ABB RobotStudio station: Final_BT19MEC092_20211026-093550.rsstn

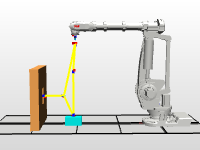
Station Solution1 (saved by RobotStudio 6.8.8307.1040)
Controller System1
  mechanical unit ROB_1: IRB6660_100_335__01, 6 joints, base frame (0, 0, 0) mm
Layout (positions relative to the parent item):
  - gripper [mechanism] at (2055.99, 1.52, 2174.48) mm, rotated rx 180 ry 0 rz 0 deg
      TCP smc_gripper at (51.61, 2.43, -191.63) mm, rotated rx 180 ry 0 rz 0 deg
      links: smc_end_effector
  - IRB6660_100_335__01 [mechanism, from Robots\IRB6660_100_335_G_01.rslib] at (0, 0, 0) mm; joint values [0.0007, 0.0004, 0, 0, 1.5708, 3.1423] (rad or m)
  - Part1 [part] at (2100, 120, 200) mm, rotated rx -90 ry 0 rz 0 deg
  - Part4 [part] at (2952.92, -603.12, 0) mm
  - Positioner_1 [smart component, from Components\Positioner.rslib] at (2100, 7, 120) mm
      properties: Object=(none); Position=[0 0 0]; Orientation=[0 0 0]; Reference=Global; ReferenceObject=(none)
  - Attacher_1 [smart component, from Components\Attacher.rslib]
      properties: Parent=gripper; Flange=0; Child=Part1; Mount=false; Offset=[0 0 0]; Orientation=[0 0 0]
  - Detacher_1 [smart component, from Components\Detacher.rslib]
      properties: Child=Part1; KeepPosition=true
  - Part11 [part] at (2800, 47, 700) mm, rotated rx 0 ry -90 rz -90 deg
  - Frame_2 [frame] at (0, 0, 197) mm
Attachment: gripper is attached to IRB6660_100_335__01 / Link6
Station signals: DI Part1_positioner
Station logic (signal -> signal, property => property):
  Solution1.Part1_positioner -> Positioner_1.Execute
  System1.at_part_1 -> Attacher_1.Execute
  System1.det_part_1 -> Detacher_1.Execute
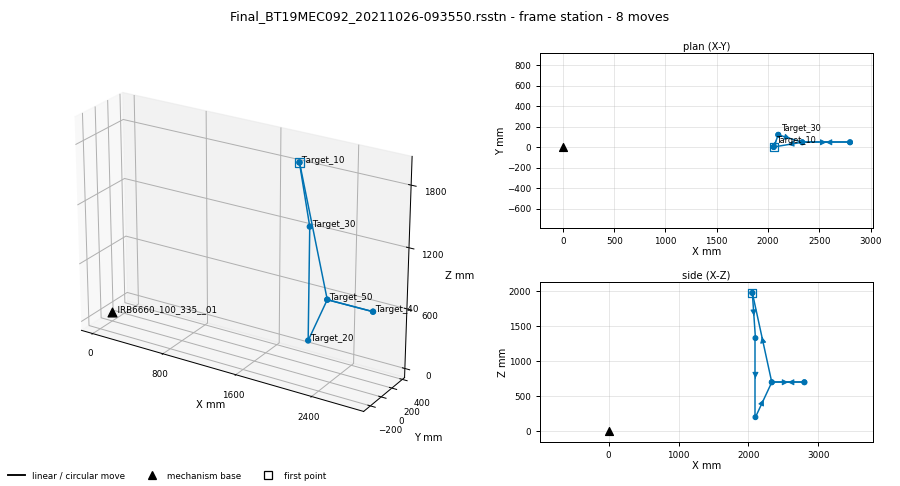
[picture p0: tool path of Final_BT19MEC092_20211026-093550.rsstn in frame station, 8 of 8 moves have a stored position in this frame; points joined in program order, loops and branches not executed]
Targets, tools, work objects and paths stored in the station, written as RAPID:
! task (no controller)
MODULE Module1
  CONST robtarget Target_20:=[[2100,120,200],[1,0,0,0],[0,0,0,0],[9E+09,9E+09,9E+09,9E+09,9E+09,9E+09]];
ENDMODULE

! task T_ROB1
MODULE CalibData
  PERS tooldata gripper:=[TRUE,[[0,0.004,197],[1,0,0,0]],[1,[0.208,-0.413,71.085],[1,0,0,0],0,0,0]];
ENDMODULE

! task T_ROB1
MODULE Module1
  CONST robtarget Target_10:=[[2055.5,0.004,1977.5],[0,0,1,0],[0,0,0,0],[9E+09,9E+09,9E+09,9E+09,9E+09,9E+09]];
  CONST robtarget Target_20:=[[2100,120,200],[0,0,1,0],[0,0,0,0],[9E+09,9E+09,9E+09,9E+09,9E+09,9E+09]];
  CONST robtarget Target_30:=[[2100,120,1331.513683654],[0,0,1,0],[0,0,0,0],[9E+09,9E+09,9E+09,9E+09,9E+09,9E+09]];
  CONST robtarget Target_40:=[[2800,47,700],[0.707106781,0,0.707106781,0],[0,-2,1,0],[9E+09,9E+09,9E+09,9E+09,9E+09,9E+09]];
  CONST robtarget Target_50:=[[2333.56728576,47,700],[0.707106781,0,0.707106781,0],[0,-2,1,0],[9E+09,9E+09,9E+09,9E+09,9E+09,9E+09]];
  CONST robtarget Target_70:=[[2055.988286208,1.517761918,1977.477993132],[0,1,0,0],[0,0,2,0],[9E+09,9E+09,9E+09,9E+09,9E+09,9E+09]];
  CONST robtarget Target_50_3:=[[2333.56728576,47,700],[0.707106781,0,0.707106781,0],[0,-2,1,0],[9E+09,9E+09,9E+09,9E+09,9E+09,9E+09]];
  PROC Path_10()
    MoveL Target_10,v100,z100,gripper\WObj:=wobj0;
    MoveL Target_30,v1000,z100,gripper\WObj:=wobj0;
    MoveL Target_20,v1000,z100,gripper\WObj:=wobj0;
    WaitTime 1;
    PulseDO at_part_1;
    MoveL Target_50,v1000,fine,gripper\WObj:=wobj0;
    MoveL Target_40,v1000,fine,gripper\WObj:=wobj0;
    WaitTime 1;
    PulseDO det_part_1;
    MoveL Target_40,v1000,z100,gripper\WObj:=wobj0;
    MoveL Target_50_3,v1000,z100,gripper\WObj:=wobj0;
    MoveL Target_70,v1000,z100,gripper\WObj:=wobj0;
  ENDPROC
ENDMODULE

